TYPE ST_XV03_CoeList :
STRUCT
	Diagnostics	: ST_Coe
END_STRUCT
END_TYPE

(* stored: Version 1.1.0.1, ProductVersion 3.1.4024.13
   DUT ST_XV03_CoeList: Id {f03682d4-52b1-05ef-127b-a4906cb737f5} *)
